PROGRAM MAIN
VAR
END_VAR

Main_Master();

END_PROGRAM

(* stored: Version 1.1.0.1, ProductVersion 3.1.4024.13
   POU MAIN: Id {b0f340cb-998b-49e4-bf91-e4e2947dabe2}, SpecialFunc None *)
